Staubli VAL3: goTo.pgx

program goTo(num x_nIndex)
  local string l_sActualTraj
  local tool l_tTool
  local bool l_bUnreached
  local string l_sMessage
  local num i
  local bool l_bContinue
  local num l_nIndexTool
  local bool l_bInside
  local bool l_bSamePoint
  local num l_nSize
  local num l_nTcpAction
  local string l_sEmpty
  local num l_nZero
  local TrajectoryItem l_tItem
begin
  // clean the movement
  if !isEmpty()
    resetMotion()
  endIf
  // get the tcp
  call trajType:getTool(l_nIndexTool)
  call saveData:getTool(l_tTool,l_nIndexTool)
  // get the trajType
  call trajType:getTrajItem(l_tItem,x_nIndex)
  // set the blend to off
  l_tItem.nom_speed.blend=off
  // AUTO ON
  if cycleStatus:nWorkingMode!=1
    // put the auto ON
    cycleStatus:bAutoON=true
    if watch(cycleStatus:bAutoON==false,3)
      l_bContinue=true
    endIf
  else
    l_bContinue=true
  endIf
  if l_bContinue
    //
    cls()
    // goTO
    call trajType:goTo(l_tTool,l_tItem.nom_speed,l_tItem.moveType,l_bUnreached,x_nIndex)
    if l_bUnreached
      // ERROR POINT NOT REACHABLE
      call language:message(l_sMessage,-5)
      call use:timerDialog(l_sMessage,1)
    else
      // GO ON
      do
        // refresh the scroll bar
        nMoveId=getMoveId()
        call use:type(0,11,toString("2",nPoint+1)+" ")
        call use:type(37,11,toString("2",x_nIndex+1)+" ")
        call use:scroll(3,11,32,abs(roundDown(nMoveId)-nMoveId)*100)
        // move to the point
        bMoveToPoint=true
        call use:typeMenu(7,"STOP")
        call showMessage()
        if !bShowMessage
          call language:message(l_sMessage,94)
          call use:timerDialog(l_sMessage+toString("",x_nIndex+1),0)
        endIf
        //
        nKey=getKey()
        delay(0)
      until (isEmpty() or nKey==255 or nKey==277)
    endIf
    //
    //look if the robot has moved
    call isAtPoint(nPoint,l_bInside)
    //DEBUT MODIF A VALIDER
    call trajType:getSizeItem(false,l_nSize)
    if nPoint<l_nSize-1
      call isAtPoint(nPoint+1,l_bSamePoint)
    endIf
    //FIN MODIF A VALIDER (+ le or l_bSamePoint)
    if !l_bInside and nPoint<x_nIndex or l_bSamePoint
      //update the nPoint
      nPoint=x_nIndex
    else
      // back position
      call isAtPoint(x_nIndex,l_bInside)
      if l_bInside and nPoint>x_nIndex
        // update the point
        nPoint=x_nIndex
      endIf
    endIf
    resetMotion()
    //
    use:bUseRefresh=true
    // clean
    bMoveToPoint=false
    call use:nullKey(nKey)
  endIf
end
